Staubli VAL3: ISBITSET.pgx

public program isBitSet(num x_value, num x_bit, bool& x_return[])
// verify if bit in num variable is set
  local string l_value
begin
  call decToBin(roundDown(x_value),l_value)
  x_return=mid(l_value,1,(len(l_value)-1)-(x_bit-1))=="1"
  if bDebug
    put("isBitSet(): "+toString("0.0",x_value)+" ? "+toString("0.0",x_bit)+" => ")
    if x_return
      putln("true")
    else
      putln("false")
    endIf
  endIf
end
